FUNCTION_BLOCK PICKER_HMI_PROXY (* Communication Unit for HMI using a plug *)
  (* Standard: 61499-2 *)
  (* Version 0.2, 2003-12-05, JHC, Rockwell Automation, Renamed from NEWCOMPFB. *)
  (* Version 0.1, 2002-01-08, JHC, Rockwell Automation, Added DLY FB as example. *)
  (* Version 0.0, 2000-05-27, JHC, Rockwell Automation *)
  (* Compiler header: package fb.rt.pnp;import fb.rt.net.*; *)
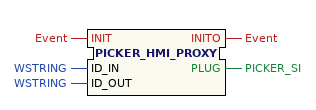
  EVENT_INPUT
    INIT; (* Initialization Request *)
  END_EVENT
  EVENT_OUTPUT
    INITO; (* Initialization Confirm *)
  END_EVENT
  VAR_INPUT
    ID_IN : WSTRING;
    ID_OUT : WSTRING;
  END_VAR
  PLUGS
    PLUG : PICKER_SI;
  END_PLUGS
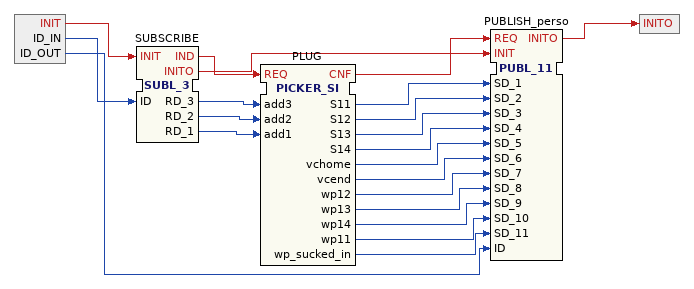
  FBS
    PUBLISH_perso : PUBL_11;
    SUBSCRIBE : SUBL_3;
  END_FBS
  EVENT_CONNECTIONS
    PLUG.CNF TO PUBLISH_perso.REQ;
    PUBLISH_perso.INITO TO INITO;
    SUBSCRIBE.IND TO PLUG.REQ;
    SUBSCRIBE.INITO TO PUBLISH_perso.INIT;
    INIT TO SUBSCRIBE.INIT;
  END_CONNECTIONS
  DATA_CONNECTIONS
    PLUG.S11 TO PUBLISH_perso.SD_1;
    PLUG.S12 TO PUBLISH_perso.SD_2;
    PLUG.S13 TO PUBLISH_perso.SD_3;
    PLUG.S14 TO PUBLISH_perso.SD_4;
    PLUG.vchome TO PUBLISH_perso.SD_5;
    PLUG.vcend TO PUBLISH_perso.SD_6;
    PLUG.wp12 TO PUBLISH_perso.SD_7;
    PLUG.wp13 TO PUBLISH_perso.SD_8;
    PLUG.wp14 TO PUBLISH_perso.SD_9;
    PLUG.wp11 TO PUBLISH_perso.SD_10;
    PLUG.wp_sucked_in TO PUBLISH_perso.SD_11;
    ID_OUT TO PUBLISH_perso.ID;
    ID_IN TO SUBSCRIBE.ID;
    SUBSCRIBE.RD_3 TO PLUG.add3;
    SUBSCRIBE.RD_2 TO PLUG.add2;
    SUBSCRIBE.RD_1 TO PLUG.add1;
  END_CONNECTIONS
END_FUNCTION_BLOCK
